// TIA Portal V20 export
FUNCTION_BLOCK "Main_Safety_RTG1"   // FB1, F_FBD
{ S7_Optimized_Access := 'TRUE' }
// stored: AutoNumber false
   VAR
      ESTOP1_Instance : ESTOP1;
   END_VAR
BEGIN

REGION Network 1
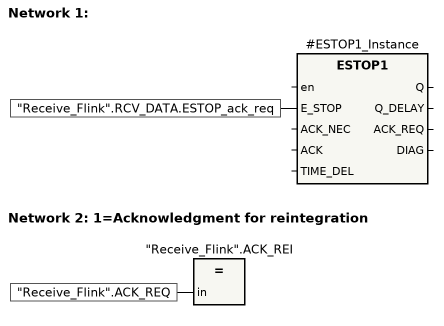
   #ESTOP1_Instance(E_STOP := "Receive_Flink".RCV_DATA.ESTOP_ack_req);   // ESTOP1
END_REGION

REGION Network 2: 1=Acknowledgment for reintegration
   "Receive_Flink".ACK_REI := "Receive_Flink".ACK_REQ;
END_REGION
END_FUNCTION_BLOCK
